VISUALIZATION Page_Alarms  // 1080x660
END_VISUALIZATION

(* stored: Version 1.1.0.1, ProductVersion 3.1.4026.13
   Visu Page_Alarms: Id {6a631766-a5bf-4017-b266-d790b30e7a5c} *)
